(* PLC project MacWin Counter, MacWin OpenPLC Compatibility Probe 1 *)
(* stored: creationDateTime 2026-07-20T00:00:00, modificationDateTime 2026-07-20T00:00:00 *)

(* Deterministic MacWin OpenPLC compatibility probe. *)
PROGRAM main
  VAR
    Counter : DINT := 0;
  END_VAR
  VAR_OUTPUT
    Pulse AT %QX0.0 : BOOL := FALSE;
  END_VAR

            Counter := Counter + 1;
Pulse := Counter >= 10;
IF Pulse THEN
  Counter := 0;
END_IF;
          
END_PROGRAM

CONFIGURATION Config0
  RESOURCE Res0 ON PLC
    TASK task0(INTERVAL := T#100ms, PRIORITY := 1);
    PROGRAM instance0 WITH task0 : main;
  END_RESOURCE
END_CONFIGURATION
